// TIA Portal V20 export
FUNCTION_BLOCK "Simulation"   // FB2, LAD
// stored: MemoryReserve 100, Namespace Unit1.Em0, SetENOAutomatically false
   VAR_INPUT
      simulation : Bool;
   END_VAR
   VAR
      instActuator { ExternalAccessible := 'False'; ExternalVisible := 'False'; ExternalWritable := 'False'} : Array[0..9] of "Simulation_Actuator";
   END_VAR
BEGIN

REGION Network 1: Two Way Actuator
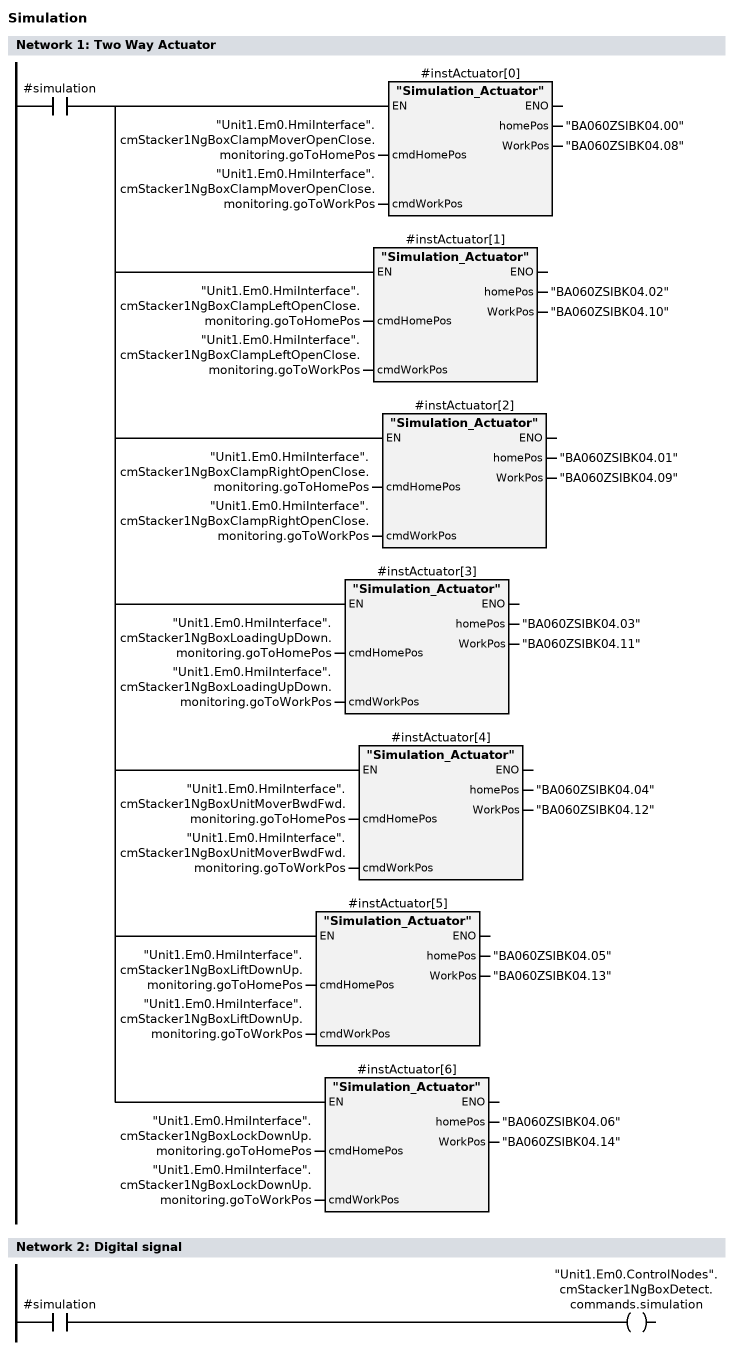
   RUNG wire#powerrail
      Contact( #simulation )
      wire#w1
      #instActuator[0](cmdHomePos := "Unit1.Em0.HmiInterface".cmStacker1NgBoxClampMoverOpenClose.monitoring.goToHomePos, cmdWorkPos := "Unit1.Em0.HmiInterface".cmStacker1NgBoxClampMoverOpenClose.monitoring.goToWorkPos, homePos => "BA060ZSIBK04.00", WorkPos => "BA060ZSIBK04.08")
   END_RUNG
   RUNG wire#w1
      #instActuator[1](cmdHomePos := "Unit1.Em0.HmiInterface".cmStacker1NgBoxClampLeftOpenClose.monitoring.goToHomePos, cmdWorkPos := "Unit1.Em0.HmiInterface".cmStacker1NgBoxClampLeftOpenClose.monitoring.goToWorkPos, homePos => "BA060ZSIBK04.02", WorkPos => "BA060ZSIBK04.10")
   END_RUNG
   RUNG wire#w1
      #instActuator[2](cmdHomePos := "Unit1.Em0.HmiInterface".cmStacker1NgBoxClampRightOpenClose.monitoring.goToHomePos, cmdWorkPos := "Unit1.Em0.HmiInterface".cmStacker1NgBoxClampRightOpenClose.monitoring.goToWorkPos, homePos => "BA060ZSIBK04.01", WorkPos => "BA060ZSIBK04.09")
   END_RUNG
   RUNG wire#w1
      #instActuator[3](cmdHomePos := "Unit1.Em0.HmiInterface".cmStacker1NgBoxLoadingUpDown.monitoring.goToHomePos, cmdWorkPos := "Unit1.Em0.HmiInterface".cmStacker1NgBoxLoadingUpDown.monitoring.goToWorkPos, homePos => "BA060ZSIBK04.03", WorkPos => "BA060ZSIBK04.11")
   END_RUNG
   RUNG wire#w1
      #instActuator[4](cmdHomePos := "Unit1.Em0.HmiInterface".cmStacker1NgBoxUnitMoverBwdFwd.monitoring.goToHomePos, cmdWorkPos := "Unit1.Em0.HmiInterface".cmStacker1NgBoxUnitMoverBwdFwd.monitoring.goToWorkPos, homePos => "BA060ZSIBK04.04", WorkPos => "BA060ZSIBK04.12")
   END_RUNG
   RUNG wire#w1
      #instActuator[5](cmdHomePos := "Unit1.Em0.HmiInterface".cmStacker1NgBoxLiftDownUp.monitoring.goToHomePos, cmdWorkPos := "Unit1.Em0.HmiInterface".cmStacker1NgBoxLiftDownUp.monitoring.goToWorkPos, homePos => "BA060ZSIBK04.05", WorkPos => "BA060ZSIBK04.13")
   END_RUNG
   RUNG wire#w1
      #instActuator[6](cmdHomePos := "Unit1.Em0.HmiInterface".cmStacker1NgBoxLockDownUp.monitoring.goToHomePos, cmdWorkPos := "Unit1.Em0.HmiInterface".cmStacker1NgBoxLockDownUp.monitoring.goToWorkPos, homePos => "BA060ZSIBK04.06", WorkPos => "BA060ZSIBK04.14")
   END_RUNG
   // the same network as SCL:
   IF #simulation THEN
       #instActuator[0](cmdHomePos := "Unit1.Em0.HmiInterface".cmStacker1NgBoxClampMoverOpenClose.monitoring.goToHomePos,   // "Simulation_Actuator"
                        cmdWorkPos := "Unit1.Em0.HmiInterface".cmStacker1NgBoxClampMoverOpenClose.monitoring.goToWorkPos,
                        homePos => "BA060ZSIBK04.00",
                        WorkPos => "BA060ZSIBK04.08");
       #instActuator[1](cmdHomePos := "Unit1.Em0.HmiInterface".cmStacker1NgBoxClampLeftOpenClose.monitoring.goToHomePos,   // "Simulation_Actuator"
                        cmdWorkPos := "Unit1.Em0.HmiInterface".cmStacker1NgBoxClampLeftOpenClose.monitoring.goToWorkPos,
                        homePos => "BA060ZSIBK04.02",
                        WorkPos => "BA060ZSIBK04.10");
       #instActuator[2](cmdHomePos := "Unit1.Em0.HmiInterface".cmStacker1NgBoxClampRightOpenClose.monitoring.goToHomePos,   // "Simulation_Actuator"
                        cmdWorkPos := "Unit1.Em0.HmiInterface".cmStacker1NgBoxClampRightOpenClose.monitoring.goToWorkPos,
                        homePos => "BA060ZSIBK04.01",
                        WorkPos => "BA060ZSIBK04.09");
       #instActuator[3](cmdHomePos := "Unit1.Em0.HmiInterface".cmStacker1NgBoxLoadingUpDown.monitoring.goToHomePos,   // "Simulation_Actuator"
                        cmdWorkPos := "Unit1.Em0.HmiInterface".cmStacker1NgBoxLoadingUpDown.monitoring.goToWorkPos,
                        homePos => "BA060ZSIBK04.03",
                        WorkPos => "BA060ZSIBK04.11");
       #instActuator[4](cmdHomePos := "Unit1.Em0.HmiInterface".cmStacker1NgBoxUnitMoverBwdFwd.monitoring.goToHomePos,   // "Simulation_Actuator"
                        cmdWorkPos := "Unit1.Em0.HmiInterface".cmStacker1NgBoxUnitMoverBwdFwd.monitoring.goToWorkPos,
                        homePos => "BA060ZSIBK04.04",
                        WorkPos => "BA060ZSIBK04.12");
       #instActuator[5](cmdHomePos := "Unit1.Em0.HmiInterface".cmStacker1NgBoxLiftDownUp.monitoring.goToHomePos,   // "Simulation_Actuator"
                        cmdWorkPos := "Unit1.Em0.HmiInterface".cmStacker1NgBoxLiftDownUp.monitoring.goToWorkPos,
                        homePos => "BA060ZSIBK04.05",
                        WorkPos => "BA060ZSIBK04.13");
       #instActuator[6](cmdHomePos := "Unit1.Em0.HmiInterface".cmStacker1NgBoxLockDownUp.monitoring.goToHomePos,   // "Simulation_Actuator"
                        cmdWorkPos := "Unit1.Em0.HmiInterface".cmStacker1NgBoxLockDownUp.monitoring.goToWorkPos,
                        homePos => "BA060ZSIBK04.06",
                        WorkPos => "BA060ZSIBK04.14");
   END_IF;
END_REGION

REGION Network 2: Digital signal
   RUNG wire#powerrail
      Contact( #simulation )
      Coil( "Unit1.Em0.ControlNodes".cmStacker1NgBoxDetect.commands.simulation )
   END_RUNG
   // the same network as SCL:
   "Unit1.Em0.ControlNodes".cmStacker1NgBoxDetect.commands.simulation := #simulation;
END_REGION

REGION Network 3 (SCL): Initializing
   IF #simulation AND "JB_Temp".Test_Homing[0] THEN
       "Unit1.Em0.HmiInterface".cmStacker1NgBoxLockDownUp.commands.commandWorkPos := true;

       "JB_Temp".Test_Homing[0] := false;
   END_IF;
END_REGION
END_FUNCTION_BLOCK
